// TIA Portal V15 export
// export: Created 2018-05-29T12:25:38.1552518Z, ExportSetting WithDefaults, DisplayName Totally Integrated Automation Portal, DisplayVersion V15, DisplayName STEP 7 Professional, DisplayVersion V15, DisplayName WinCC Professional, DisplayVersion V15, DisplayName TIA Portal Openness, DisplayVersion V15
FUNCTION "P101_fc" : Void   // FC1, STL
TITLE = P101_fc
{ S7_Optimized_Access := 'TRUE' }
VERSION : 0.1
// test
// stored: AutoNumber true, UDAEnableTagReadback false
BEGIN

NETWORK
TITLE = Main
// comment: PLC1


// Call the CM FB with the corresponding DB instance
      CALL  "BST_MOTOR_400", "P101"
      ( AUTO_ON    := ,
        L_AUT      := ,
        FB_ON      := ,
        ERR_EXTERN := ,
        QRUN       := ,
        QSTOP      := ,
        QCMD_ON    := ,
        QMON_ERR   := ,
        QMPS       := ,
        QERR       := 
      );
END_FUNCTION
